// TIA Portal V19 export
DATA_BLOCK "A0302_Centratori"   // DB110
// stored: InstanceOfName A0302_Centratori_FB, InstanceOfType FB
"A0302_Centratori_FB"
   // VAR_INPUT
   //    AreaInterface : "AreaInterface";
   //    ZSI : "udt_ZoneSafetyInterface";
   //    DSI : "udt_DeviceSafetyInterface";
   //    DataIn : Struct
   //       OP : "OP_PB";
   //    END_STRUCT;
   //    CIn : Struct
   //       Manager : Struct
   //          Sollevamento : "ValveMachine_Manager";
   //          Centraggio : "ValveMachine_Manager";
   //       END_STRUCT;
   //       SemiAut_Pb : Bool;
   //       Rulliera : Struct
   //          Coda : Struct
   //             Sens : Struct
   //                FTC_Rall : Bool;
   //                FTC_Prox_Ing : Bool;
   //             END_STRUCT;
   //          END_STRUCT;
   //          Centro : Struct
   //             Sens : Struct
   //                FTC_Centrale : Bool;
   //             END_STRUCT;
   //          END_STRUCT;
   //       END_STRUCT;
   //       CarroPareggCoda : Struct
   //          Ax : "Positioning_DOL_Machine_COut";
   //          Bloccaggio : "ValveMachine_COut";
   //          BattutaVerticale : "ValveMachine_COut";
   //          PareggiatoreLong : "ValveMachine_COut";
   //          Sens : Struct
   //             FTC_Ingombro_In : Bool;
   //             FTC_Ingombro_Out : Bool;
   //             PresenzaMat : Bool;
   //          END_STRUCT;
   //       END_STRUCT;
   //       CarroPareggTesta : Struct
   //          Ax : "Positioning_DOL_Machine_COut";
   //          Bloccaggio : "ValveMachine_COut";
   //          Centraggio : "ValveMachine_COut";
   //          Sollevatore : "ValveMachine_COut";
   //          Sens : Struct
   //             FTC1_Rall : Bool;
   //             FTC2_Prox_Ls : Bool;
   //             PresenzaMat : Bool;
   //          END_STRUCT;
   //       END_STRUCT;
   //       BTrk : Struct
   //          ZoneA0302Entry_Empty : Bool;
   //          ZoneA0302Exit_Empty : Bool;
   //       END_STRUCT;
   //    END_STRUCT;
   //    Config : Struct
   //       Centraggio : Array[1..3] of "ValveMachine_Config";
   //       Sollevamento : Array[1..3] of "ValveMachine_Config";
   //       DelayMissingCondition : Time;
   //       WorkWindows : Struct
   //          Coda : Struct
   //             Min : LReal;
   //             Max : LReal;
   //          END_STRUCT;
   //          Testa : Struct
   //             Min : LReal;
   //             Max : LReal;
   //          END_STRUCT;
   //       END_STRUCT;
   //    END_STRUCT;
   // END_VAR
   // VAR_OUTPUT
   //    MachineInterface : "MachineInterface";
   //    COut : Struct
   //       Centratori : "ValveMachine_COut";
   //       Centraggio : "ValveMachine_COut";
   //       Sollevamento : "ValveMachine_COut";
   //    END_STRUCT;
   // END_VAR
   // VAR
   //    Alarm : Struct
   //       Centraggio : Array[1..3] of "ValveAlr";
   //       Sollevamento : Array[1..3] of "ValveAlr";
   //    END_STRUCT;
   //    Warning : Struct
   //       Centratore : Array[1..3] of "ValveMachine_Wng";
   //       Sollevamento : Array[1..3] of "ValveMachine_Wng";
   //       OP_REST_Centr_MissingCnd : Bool;
   //       OP_WORK_Centr_MissingCnd : Bool;
   //       OP_REST_Sollev_MissingCnd : Bool;
   //       OP_WORK_Sollev_MissingCnd : Bool;
   //    END_STRUCT;
   //    HMI : Struct
   //       Selection : Struct
   //          Centraggio : Array[1..3] of Bool;
   //          Sollevamento : Array[1..3] of Bool;
   //       END_STRUCT;
   //       Centratori_Sts : "UDT_HMI-Sts_ValvePosA0301";
   //       Centraggio_Sts { S7_SetPoint := 'True'} : "UDT_HMI-Sts_ValvePosA0301";
   //       Sollevamento_Sts { S7_SetPoint := 'True'} : "UDT_HMI-Sts_ValvePosA0301";
   //    END_STRUCT;
   //    Centraggio : Array[1..3] of "ValveMachine_FB";
   //    Sollevamento { S7_SetPoint := 'True'} : Array[1..3] of "ValveMachine_FB";
   //    Sts : Struct
   //       Centraggio : Struct
   //          OP_Rest_Cnd : Bool;
   //          Op_Work_Cnd : Bool;
   //       END_STRUCT;
   //       Sollevamento : Struct
   //          OP_Rest_Cnd : Bool;
   //          Op_Work_Cnd : Bool;
   //       END_STRUCT;
   //       Centratori_Alarm : Bool;
   //       Centraggio_AlarmPresence : Bool;
   //       Sollevamento_AlarmPresence : Bool;
   //       OP_CanMoveFreely : Bool;
   //    END_STRUCT;
   //    Ctrl : Struct
   //       Centraggio : Struct
   //          OP_Rest_Man : Bool;
   //          OP_Work_Man : Bool;
   //          OP_Rest_Aut : Bool;
   //          OP_Work_Aut : Bool;
   //          OP_Rest : Bool;
   //          OP_Work : Bool;
   //       END_STRUCT;
   //       Sollevamento : Struct
   //          OP_Rest_Man : Bool;
   //          OP_Work_Man : Bool;
   //          OP_Rest_Aut : Bool;
   //          OP_Work_Aut : Bool;
   //          OP_Rest : Bool;
   //          OP_Work : Bool;
   //       END_STRUCT;
   //    END_STRUCT;
   //    AUX : Struct
   //       Centraggio : Struct
   //          OP_Rest_PB : Bool;
   //          OP_Work_PB : Bool;
   //       END_STRUCT;
   //       Sollevamento : Struct
   //          OP_Rest_PB : Bool;
   //          OP_Work_PB : Bool;
   //       END_STRUCT;
   //    END_STRUCT;
   //    TON_OP_REST_Centr_MissingCnd { S7_SetPoint := 'True'} : TON_TIME;
   //    TON_OP_WORK_Centr_MissingCnd { S7_SetPoint := 'True'} : TON_TIME;
   //    TON_OP_REST_Sollev_MissingCnd { S7_SetPoint := 'True'} : TON_TIME;
   //    TON_OP_WORK_Sollev_MissingCnd { S7_SetPoint := 'True'} : TON_TIME;
   //    DelayMissingCondition : Time;
   //    TON_Anticipi : Struct
   //       Work : Struct
   //          Sollevamento : Array[1..3] of IEC_TIMER;
   //          Centraggio : Array[1..3] of IEC_TIMER;
   //       END_STRUCT;
   //       Rest : Struct
   //          Sollevamento : Array[1..3] of IEC_TIMER;
   //          Centraggio : Array[1..3] of IEC_TIMER;
   //       END_STRUCT;
   //    END_STRUCT;
   // END_VAR
BEGIN
   HMI.Selection.Centraggio[1..3] := TRUE;
   HMI.Selection.Sollevamento[1..3] := TRUE;
END_DATA_BLOCK
